{attribute 'enable_dynamic_creation'}
FUNCTION_BLOCK FutureMCSetPosition EXTENDS FB_AbstructFuture
VAR_INPUT
END_VAR
VAR_OUTPUT
END_VAR
VAR
	_fb_set_position	: MC_SetPosition;
	_axis: REFERENCE TO AXIS_REF;
	_position	: MC_LREAL;
	_mode		: BOOL;
	_option 	: ST_SetPositionOptions;
	_error_id :UDINT;
	_exec_state : UDINT;
END_VAR

METHOD abort : BOOL // Return TRUE if finish.
END_METHOD

METHOD execute : BOOL // Return TRUE if finish.

CASE _exec_state OF
	0:
		_fb_set_position( Axis:= _axis, Execute := FALSE);
		_fb_set_position(
				Axis := _axis,
				Execute := TRUE, 
				Position := _position,
				Mode := _mode,
				Options := _option
		);
		_exec_state := 1;
	1:
		IF _fb_set_position.Busy THEN
			_fb_set_position( Axis:= _axis, Execute := FALSE);
		END_IF
END_CASE

_error_id := _fb_set_position.ErrorID;
execute := _fb_set_position.Done OR _fb_set_position.Error;
END_METHOD

METHOD init : BOOL // Return TRUE if finish.
_exec_state := 0;
init := TRUE;
END_METHOD

PROPERTY nErrorID : UDINT
GET
nErrorID := _error_id;
END_GET
SET
END_SET
END_PROPERTY

METHOD set_options : BOOL
VAR_INPUT
	mode		: BOOL;
	option 	: ST_SetPositionOptions;
END_VAR
_mode := mode;
_option := option;
END_METHOD

METHOD set_parameters : BOOL
VAR_INPUT
	axis: REFERENCE TO AXIS_REF;
	position	: MC_LREAL;
END_VAR
_axis REF= axis;
_position := position;
END_METHOD

END_FUNCTION_BLOCK

(* stored: Version 1.1.0.1, ProductVersion 3.1.4024.12
   POU FutureMCSetPosition: Id {d61bff14-9e58-4f9b-b583-353e0d0667c2}, SpecialFunc None
   Method abort: Id {e6c82ab6-3275-49eb-8d56-5c988eed9a96}
   Method execute: Id {6e6f1e42-98ad-4c1b-b340-999b8148b2fe}
   Method init: Id {20b0fd3a-f8ec-456d-a95d-c961ca55e36b}
   Property nErrorID: Id {fef29eb0-8ad6-4992-85bd-77e274eb424f}
   Get Get: Id {0dff01db-06ac-495c-b6df-d8ea0fdd89b7}
   Set Set: Id {4464918e-fa0d-4365-85fa-d4a5a40de5ec}
   Method set_options: Id {b7b03d5a-6cb0-4d9b-9472-cf91ae3da253}
   Method set_parameters: Id {fa949765-5486-4de3-b42b-76d600f91797} *)
